{attribute 'qualified_only'}
{attribute 'strict'}
TYPE E_StationBufferState :
(
	Idle := 0,
	CheckBuffer,
	StartMove,
	WaitMove
	
);
END_TYPE

(* stored: Version 1.1.0.1, ProductVersion 3.1.4024.2
   DUT E_StationBufferState: Id {407dc16a-cc0d-4750-9322-8078f0c6b160} *)
